(* CODESYS project Турникет.project

Project tree, tasks and I/O mapping:
  Device : CODESYS Control Win V3 x64, 3S - Smart Software Solutions GmbH, version 3.5.11.0
    application Application
      libraries: Standard, * (System); VisuDialogs, * (System)
      task MainTask (cyclic, interval t#20ms, priority 1) calls Controller
      task VISU_TASK (cyclic, interval 100 ms, priority 31) calls VisuElems.Visu_Prg
      task Plant_task (cyclic, interval t#20ms, priority 1) calls Plant
      program Controller [ST]
      global variables GVL
      visualisation Visualization
      program Plant [ST]
      image pool ImagePool
  libraries: VisuSymbols, 3.5.10.0 (System)
  text list GlobalTextList
  5ce3da45-db07-42e7-a21c-a00fff4ed8f6|Assets\exit.jpeg
  5ce3da45-db07-42e7-a21c-a00fff4ed8f6|Assets\to_trains.jpg
  5ce3da45-db07-42e7-a21c-a00fff4ed8f6|Assets\men.jpg
  text list System
*)

// Device/Application/GVL
VAR_GLOBAL

    // ─────────────────────────────
    // Environment (кнопки симуляции)
    // ─────────────────────────────
    simPersonForward     : BOOL;
    simPersonBackward    : BOOL;
    simJump              : BOOL;

    resetButton          : BOOL;
    forceClose           : BOOL;


    // ─────────────────────────────
    // Sensors
    // ─────────────────────────────
    sensorExit1          : BOOL;
    sensorExit2          : BOOL;
    sensorExit3          : BOOL;

    weightSensor1        : BOOL;
    weightSensor2        : BOOL;


    // ─────────────────────────────
    // Actuators
    // ─────────────────────────────
    openGate             : BOOL;
    closeGate            : BOOL;
    buzzerAlarm          : BOOL;


    // ─────────────────────────────
    // Plant states
    // ─────────────────────────────
    gatePosition         : REAL := 100.0; // 100=open
    personPosition       : REAL := -50.0;

	// Центры двух створок для визуализации
    gateLeftCenter  : REAL := 80;
	gateRightCenter : REAL := 78;
	
	gateLeftY       : REAL := 0;
	gateRightY      : REAL := 95;
	
	// Для стопа перед створками
	passingForward  : BOOL;
    passingBackward : BOOL;
	
	gateLineBackward : REAL := 845.0;
	gateLineForward : REAL := 200.0;
	personWidth      : REAL := 295.0;
	gateLineX        : REAL := 845.0;
	gatePassPos      : REAL := 80.0;
	
END_VAR

// Device/Application/Controller
PROGRAM Controller
VAR
    // Последовательность корректного прохода
    sequenceStep : INT := 0;   // 0-ждём 1, 1-ждём 2, 2-ждём 3

    // Предыдущие состояния датчиков и детекция некорректного прохода
    prev1 : BOOL;
    prev2 : BOOL;
    prev3 : BOOL;
	
	reversePending2 : BOOL;
	reversePending3 : BOOL;
	
	reverseTimer2 : TON;
	reverseTimer3 : TON;

    // Триггер кнопки сброса
    resetTrig : R_TRIG;
	resetOverride : BOOL;

    // Таймеры "зависших" датчиков
    timer1 : TON;
    timer2 : TON;
    timer3 : TON;
    timerW1 : TON;
    timerW2 : TON;
	
	// Для отображения
	timer1_sec : REAL;
	timer2_sec  : REAL;
	timer3_sec  : REAL;
	timerW1_sec : REAL;
	timerW2_sec : REAL;

    // Состояния системы
	intrusionAlarm   : BOOL := FALSE;  // нарушение направления, закрытие + сирена
	weightAlarm      : BOOL := FALSE;  // датчики веса, только сирена
	stuckAlarm       : BOOL := FALSE;  // датчик завис >30 c, только сирена
	forcedCloseActive: BOOL := FALSE;  // режим принудительного закрытия
END_VAR

// ======================================================
// 1. Детектор фронта кнопки Reset
// ======================================================
resetTrig(CLK := resetButton);


// ======================================================
// 2. Reset имеет высокий приоритет
// ======================================================
IF resetTrig.Q THEN
    resetOverride := TRUE;

    intrusionAlarm := FALSE;
    weightAlarm := FALSE;
    stuckAlarm := FALSE;
    forcedCloseActive := FALSE;
    sequenceStep := 0;

    prev1 := FALSE;
    prev2 := FALSE;
    prev3 := FALSE;

    reversePending2 := FALSE;
    reversePending3 := FALSE;
END_IF;


// ======================================================
// 3. Автоматическое снятие resetOverride
// ======================================================
IF resetOverride AND
   NOT sensorExit1 AND
   NOT sensorExit2 AND
   NOT sensorExit3 AND
   NOT weightSensor1 AND
   NOT weightSensor2 THEN
    resetOverride := FALSE;
END_IF;


// ======================================================
// 4. Принудительное закрытие оператором
// ======================================================
IF forceClose AND NOT resetOverride THEN
    forcedCloseActive := TRUE;
END_IF;


// ======================================================
// 5. Таймеры зависших датчиков
// ======================================================
timer1(IN := sensorExit1 AND NOT resetOverride, PT := T#30S);
timer2(IN := sensorExit2 AND NOT resetOverride, PT := T#30S);
timer3(IN := sensorExit3 AND NOT resetOverride, PT := T#30S);
timerW1(IN := weightSensor1 AND NOT resetOverride, PT := T#30S);
timerW2(IN := weightSensor2 AND NOT resetOverride, PT := T#30S);

// Короткие таймеры подтверждения обратного прохода
reverseTimer2(IN := reversePending2, PT := T#2.5S);
reverseTimer3(IN := reversePending3, PT := T#2.5S);

// Значения для визуализации
timer1_sec := TIME_TO_DINT(timer1.ET) / 1000.0;
timer2_sec := TIME_TO_DINT(timer2.ET) / 1000.0;
timer3_sec := TIME_TO_DINT(timer3.ET) / 1000.0;
timerW1_sec := TIME_TO_DINT(timerW1.ET) / 1000.0;
timerW2_sec := TIME_TO_DINT(timerW2.ET) / 1000.0;

// ======================================================
// 6. Залипание датчиков
// ======================================================
IF NOT resetOverride THEN
    IF timer1.Q OR timer2.Q OR timer3.Q OR timerW1.Q OR timerW2.Q THEN
        stuckAlarm := TRUE;
    END_IF;
END_IF;

// ======================================================
// 7. Проверка нарушений
// ======================================================
IF NOT resetOverride AND NOT intrusionAlarm AND NOT forcedCloseActive AND NOT stuckAlarm THEN

    // Попытка перепрыгнуть / опора на корпус
    IF weightSensor1 AND weightSensor2 THEN
        weightAlarm := TRUE;
    END_IF;

    // Подозрение на обратный проход
    IF (sequenceStep = 0) AND sensorExit2 AND NOT prev2 THEN
        reversePending2 := TRUE;
    END_IF;

    IF (sequenceStep = 0) AND sensorExit3 AND NOT prev3 THEN
        reversePending3 := TRUE;
    END_IF;

    // Подтверждение обратного прохода
    IF reversePending2 AND sensorExit1 THEN
        intrusionAlarm := TRUE;
        reversePending2 := FALSE;
    END_IF;

    IF reversePending3 AND (sensorExit2 OR sensorExit1) THEN
        intrusionAlarm := TRUE;
        reversePending3 := FALSE;
    END_IF;

    // Истечение окна подтверждения
    IF reverseTimer2.Q THEN
        reversePending2 := FALSE;
    END_IF;

    IF reverseTimer3.Q THEN
        reversePending3 := FALSE;
    END_IF;

    // Нарушение порядка внутри нормальной последовательности
    IF (sequenceStep = 1) AND sensorExit3 AND NOT prev3 THEN
        intrusionAlarm := TRUE;
    END_IF;

END_IF;

// ======================================================
// 8. Конечный автомат корректного прохода
// ======================================================
IF NOT resetOverride AND NOT intrusionAlarm AND NOT weightAlarm AND NOT stuckAlarm AND NOT forcedCloseActive THEN

    CASE sequenceStep OF

        0:
            IF sensorExit1 AND NOT prev1 THEN
                sequenceStep := 1;
            END_IF;

        1:
            IF sensorExit2 AND NOT prev2 THEN
                sequenceStep := 2;
            END_IF;

        2:
            IF sensorExit3 AND NOT prev3 THEN
                sequenceStep := 3;
            END_IF;

        3:
            IF NOT sensorExit1 AND NOT sensorExit2 AND NOT sensorExit3 THEN
                sequenceStep := 0;
            END_IF;

    END_CASE;

END_IF;


// ======================================================
// 9. Формирование выходных сигналов
// ======================================================
openGate := FALSE;
closeGate := FALSE;
buzzerAlarm := FALSE;

IF resetOverride THEN
    openGate := TRUE;
    closeGate := FALSE;
    buzzerAlarm := FALSE;

ELSIF forcedCloseActive THEN
    closeGate := TRUE;

ELSIF intrusionAlarm THEN
    closeGate := TRUE;
    buzzerAlarm := TRUE;

ELSIF weightAlarm OR stuckAlarm THEN
    buzzerAlarm := TRUE;

ELSE
    openGate := TRUE;
END_IF;


// ======================================================
// 10. Гарантия взаимного исключения команд
// ======================================================
IF closeGate THEN
    openGate := FALSE;
END_IF;


// ======================================================
// 11. Сохранение предыдущих состояний
// ======================================================
prev1 := sensorExit1;
prev2 := sensorExit2;
prev3 := sensorExit3;

END_PROGRAM

// Device/Application/Plant
PROGRAM Plant
VAR
    // Скорости моделирования
    personSpeed : REAL := 2.0;
    gateSpeed   : REAL := 5.0;

    // Внутренние переменные для управления движением
    moveForward : BOOL;
    moveBackward: BOOL;
	gateIsOpen: BOOL;
	simHoldS1: BOOL;
	simHoldS2: BOOL;
	simHoldS3: BOOL;
	simHoldW1: BOOL;
	simHoldW2: BOOL;
END_VAR

// ======================================================
// 1. Управление движением человека
// ======================================================

// Кнопка "Нормальный проход" запускает движение из PAID_AREA в FREE_AREA
IF simPersonForward THEN
    moveForward := TRUE;
END_IF;

// Кнопка "Обратный проход" запускает движение из FREE_AREA в PAID_AREA
IF simPersonBackward THEN
    moveBackward := TRUE;
END_IF;

// Взаимное исключение направлений
IF moveForward THEN
    moveBackward := FALSE;
END_IF;

IF moveBackward THEN
    moveForward := FALSE;
END_IF;



// ======================================================
// 2. Перемещение человека с учётом закрытых створок
// ======================================================

IF passingForward THEN
    passingBackward := FALSE;
END_IF;

IF passingBackward THEN
    passingForward := FALSE;
END_IF;

IF moveForward THEN
    personPosition := personPosition + personSpeed;
END_IF;

IF moveBackward THEN
    personPosition := personPosition - personSpeed;
END_IF;

// ======================================================
// 3. Автоматическое завершение прохода
// ======================================================

// Человек полностью вышел в FREE_AREA
IF personPosition > 950.0 THEN
    personPosition := 170.0;
    moveForward := FALSE;
END_IF;

// Человек полностью вернулся в PAID_AREA
IF personPosition < 170.0 THEN
    personPosition := 950.0;
    moveBackward := FALSE;
END_IF;


// ======================================================
// 4. Моделирование оптических датчиков
// ======================================================

IF simHoldS1 THEN
    sensorExit1 := TRUE;
ELSE
    sensorExit1 :=
        (personPosition >= 400.0) AND
        (personPosition <= 430.0);
END_IF;

IF simHoldS2 THEN
    sensorExit2 := TRUE;
ELSE
	sensorExit2 :=
		(personPosition >= 600.0) AND
		(personPosition <= 630.0);
END_IF;

IF simHoldS3 THEN
    sensorExit3 := TRUE;
ELSE
	sensorExit3 :=
		(personPosition >= 800.0) AND
		(personPosition <= 830.0);
END_IF;

// ======================================================
// 5. Моделирование датчиков веса
// ======================================================

// Кнопка simJump имитирует попытку перелезть через турникет
weightSensor1 := simHoldW1 OR simJump;
weightSensor2 := simHoldW2 OR simJump;

// ======================================================
// 6. Анимация створок
// ======================================================

// gatePosition:
// 100.0 = полностью открыты
//   0.0 = полностью закрыты

IF openGate THEN
    gatePosition := gatePosition + gateSpeed;
END_IF;

IF closeGate THEN
    gatePosition := gatePosition - gateSpeed;
END_IF;


// Ограничение диапазона
IF gatePosition > 100.0 THEN
    gatePosition := 100.0;
END_IF;

IF gatePosition < 0.0 THEN
    gatePosition := 0.0;
END_IF;


// ======================================================
// 7. Логический индикатор состояния створок
// ======================================================

gateIsOpen := (gatePosition >= 99.0);

// Закрытое состояние:
// левая створка  -> центр 835
// правая створка -> центр 998
// Полностью открытое состояние даёт проём 312 px

// Центры створок
gateLeftCenter  := 80.0 - (gatePosition * 1.53);
gateRightCenter := 75.0 + (gatePosition * 1.53);

// Левые координаты прямоугольников для визуализации
gateLeftY := gateLeftCenter - 78.5;
gateRightY := gateRightCenter - 78.5;


// ======================================================
// 8. Автоматический сброс кнопок симуляции
// ======================================================

// Чтобы кнопки работали как "импульсные", а не как переключатели
IF simPersonForward THEN
    simPersonForward := FALSE;
END_IF;

IF simPersonBackward THEN
    simPersonBackward := FALSE;
END_IF;

END_PROGRAM

// Device/Application/Visualization
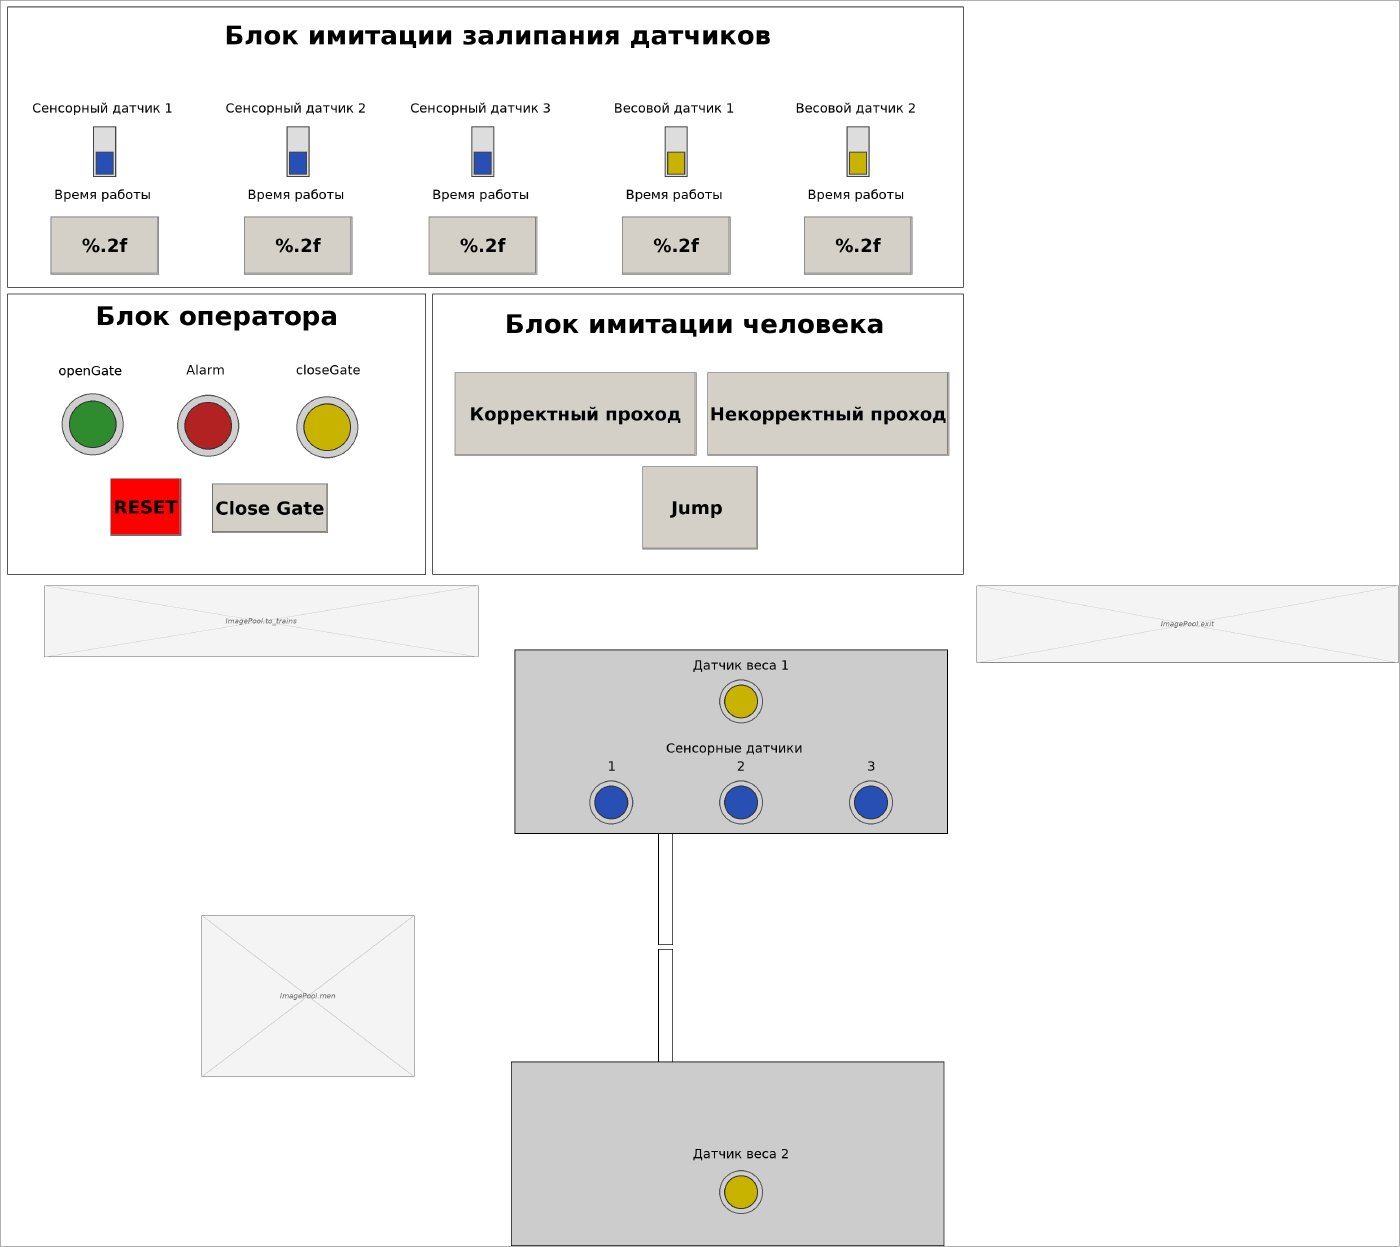
VISUALIZATION Visualization  // 1940x1728
    Rectangle (10,407 580x389)
    Rectangle (599,407 736x389)
    Rectangle (10,9 1325x389)
    Rectangle (912,1315 20x157)
        p2738717112: gateRightY
    Rectangle (912,1152 20x157)
        p2738717112: gateLeftY
    Lamp1 (79,538 99x100), variable: openGate, style: Lamp-Lamp1-Green
    Lamp1 (404,542 99x100), variable: closeGate, style: Lamp-Lamp1-Yellow
    Lamp1 (239,540 99x100), variable: buzzerAlarm, style: Lamp-Lamp1-Red
    Button (153,663 98x79), "RESET"
        OnMouseDown:  ToggleVariable=resetButton
        OnMouseUp:  ToggleVariable=resetButton
    Label (50,499 150x30), "openGate"
    Label (210,498 150x30), "Alarm"
    Label (380,498 150x30), "closeGate"
    Rectangle (713,900 600x255)
    Rectangle (708,1471 600x255)
    Image (279,1268 295x224), angle 270, image: ImagePool.men
        p3560616238: personPosition
    Button (630,516 335x115), "Корректный проход"
        OnMouseDown:  ToggleVariable=simPersonForward
    Button (980,516 335x115), "Некорректный проход"
        OnMouseDown:  ToggleVariable=simPersonBackward
    Image (1353,811 585x107), image: ImagePool.exit
    Image (61,811 602x99), image: ImagePool.to_trains
    Lamp1 (812,1077 70x70), variable: sensorExit1, style: Lamp-Lamp1-Blue
    Lamp1 (992,1077 70x70), variable: sensorExit2, style: Lamp-Lamp1-Blue
    Lamp1 (1172,1077 70x70), variable: sensorExit3, style: Lamp-Lamp1-Blue
    Button (294,670 160x68), "Close Gate"
        OnMouseDown:  ToggleVariable=forceClose
        OnMouseUp:  ToggleVariable=forceClose
    Button (890,646 160x115), "Jump"
        OnMouseDown:  ToggleVariable=simJump
        OnMouseUp:  ToggleVariable=simJump
    Lamp1 (992,937 70x70), variable: weightSensor1, style: Lamp-Lamp1-Yellow
    Lamp1 (992,1617 70x70), variable: weightSensor2, style: Lamp-Lamp1-Yellow
    Label (952,907 150x30), "Датчик веса 1"
    Label (952,1584 150x30), "Датчик веса 2"
    Label (751,1052 194x20), "1"
    Label (933,1052 188x20), "2"
    Label (1112,1052 191x20), "3"
    Button (70,300 150x80), "%.2f", text variable: Controller.timer1_sec
    DipSwitch (110,175 70x70), variable: Plant.simHoldS1, behaviour: TOGGLE, style: Switch-DipSwitch-Blue
    Label (30,135 224x30), "Сенсорный датчик 1"
    Label (30,255 224x30), "Время работы"
    Button (338,300 150x80), "%.2f", text variable: Controller.timer2_sec
    DipSwitch (378,175 70x70), variable: Plant.simHoldS2, behaviour: TOGGLE, style: Switch-DipSwitch-Blue
    Label (298,135 224x30), "Сенсорный датчик 2"
    Label (298,255 224x30), "Время работы"
    Button (594,300 150x80), "%.2f", text variable: Controller.timer3_sec
    DipSwitch (634,175 70x70), variable: Plant.simHoldS3, behaviour: TOGGLE, style: Switch-DipSwitch-Blue
    Label (554,135 224x30), "Сенсорный датчик 3"
    Label (554,255 224x30), "Время работы"
    Button (862,300 150x80), "%.2f", text variable: Controller.timerW1_sec
    DipSwitch (902,175 70x70), variable: Plant.simHoldW1, behaviour: TOGGLE, style: Switch-DipSwitch-Yellow
    Label (822,135 224x30), "Весовой датчик 1"
    Label (822,255 224x30), "Время работы"
    Button (1114,300 150x80), "%.2f", text variable: Controller.timerW2_sec
    DipSwitch (1154,175 70x70), variable: Plant.simHoldW2, behaviour: TOGGLE, style: Switch-DipSwitch-Yellow
    Label (1074,135 224x30), "Весовой датчик 2"
    Label (1074,255 224x30), "Время работы"
    Label (222,29 936x40), "Блок имитации залипания датчиков"
    Label (93,418 415x40), "Блок оператора"
    Label (681,429 563x40), "Блок имитации человека"
    Label (902,1027 231x20), "Сенсорные датчики"
END_VISUALIZATION

(* text list System (id | default)
  Apr | Apr
  April | April
  Aug | Aug
  August | August
  Dec | Dec
  December | December
  Feb | Feb
  February | February
  Fri | Fri
  Friday | Friday
  Jan | Jan
  January | January
  Jul | Jul
  July | July
  Jun | Jun
  June | June
  Mar | Mar
  March | March
  May | May
  May_3Letter | May
  Mon | Mon
  Monday | Monday
  Nov | Nov
  November | November
  Oct | Oct
  October | October
  Sat | Sat
  Saturday | Saturday
  Sep | Sep
  September | September
  Sun | Sun
  Sunday | Sunday
  Thu | Thu
  Thursday | Thursday
  Tue | Tue
  Tuesday | Tuesday
  Wed | Wed
  Wednesday | Wednesday
   |  *)
